Fanuc KAREL source: kt00490.KL

-- PROVISIONAL review KL for V770-1; original PC SHA256 2c65728d445cee5e522dc9f6f4ce9545070c1591a0372daad5ac74e15a0e0f4b
-- Incomplete behavior may be omitted. Consult companion uncertainty JSON. Do not deploy.
PROGRAM KT00490
%NOLOCKGROUP
-- UNRESOLVED_DECL P1 type=000101
-- UNRESOLVED_DECL P2 type=000199
-- UNRESOLVED_DECL OUT type=000102
BEGIN
  -- UNRESOLVED_PC offsets 5-39; opcodes 49,49,7E,60,7E,4A
  -- UNRESOLVED_PC offsets 44-48; opcodes 7F
END KT00490
